INTERFACE I_Base EXTENDS SYSTEM.__QUERYINTERFACE

END_INTERFACE

(* stored: Version 1.1.0.1, ProductVersion 3.1.4026.18
   Itf I_Base: Id {8828ad51-d726-4f54-b5de-d78b11ab1abf} *)
